(* PLC project CODESYS_HashTable_Struct_Example.project, CODESYS CODESYS V3.5 SP20 Patch 3 *)
(* stored: creationDateTime 2025-01-24T23:29:18.215425, modificationDateTime 2025-01-24T23:25:16.619379 *)

TYPE ST_Product : STRUCT
  id : STRING;  (* 製品ID *)
  name : STRING;  (* 製品名 *)
  width : UINT;  (* 幅 *)
  length : UINT;  (* 長さ *)
  height : UINT;  (* 高さ *)
END_STRUCT;
END_TYPE

(* values of E_ProductSettingState: Create: 新規作成; Edit: 編集 *)

{attribute 'qualified_only'}
{attribute 'strict'}
TYPE E_ProductSettingState : (Initial := 0, Create, Edit);
END_TYPE

INTERFACE IProductElement
PROPERTY ProductValue : ST_Product
END_PROPERTY
END_INTERFACE

PROGRAM PRG_ProductSetting
  VAR
    HashTableFactory : COL.HashTableFactory;  (* Factory to create a hash table on heap memory. *)
    productMap : COL.IMap3 := HashTableFactory.Create(udiMaxElements := 100);  (* Creates a hashtable on heap memory. NOTE: Collections that have been created with this Factory are not online change safe. *)
    productElementFactory : FB_ProductElementFactory;
    productNameArray : ARRAY[0..GVL.MAX_PRODUCT_NUM] OF STRING;  (* Visualizaton用 *)
    pnArrayLastIndex : UINT := 0;  (* 次に挿入する位置 *)
    state : E_ProductSettingState := E_ProductSettingState.Initial;
    selectedProductIndex : UINT;
    selectedProductId : STRING;
    visuProduct : ST_Product;
    msgBoxMessage : STRING;  (* メッセージBOX用 *)
    msgBoxEnabled : BOOL;
    msgBoxTap : BOOL;
    tmpValues : ARRAY[0..GVL.MAX_PRODUCT_NUM] OF ST_Product;  (* デバッグ用 *)
    iterator : COL.ListIterator;
    itfElement : COL.IElement;
    itfProductElement : IProductElement;
    xResult : BOOL;
    i : UINT;  (* 一時変数 *)
  END_VAR

                    //デバッグ用
i:=0;
productMap.Values(iterator);
WHILE iterator.HasNext() DO
	iterator.Next(itfElement=>itfElement);
	xResult := __QUERYINTERFACE(itfElement, itfProductElement);
	tmpValues[i] := itfProductElement.ProductValue;
	i:=i+1;
END_WHILE

//メッセージBOXを閉じる
IF msgBoxTap THEN
	msgBoxEnabled := FALSE;
	msgBoxTap := FALSE;
END_IF


//現在状態ごとの処理
IF state = E_ProductSettingState.Initial AND pnArrayLastIndex <> 0 THEN
	selectedProductIndex := 0;
	UpdateSelectedProduct();
	state := E_ProductSettingState.Edit;
END_IF
	

                  

METHOD DeleteProductFromNameArray
  VAR_INPUT
    info : ST_Product;
  END_VAR
  VAR
    i : UINT;
    deleteIndex : UINT;
    productId : STRING;
  END_VAR
                          IF pnArrayLastIndex > GVL.MAX_PRODUCT_NUM THEN
	RETURN;
END_IF


IF pnArrayLastIndex <> 0 THEN
	//昇順にソートされている前提で挿入個所を探索する
	FOR deleteIndex:=0 TO pnArrayLastIndex-1 DO
		productId := GetIdFromProductName(ADR(productNameArray[deleteIndex]));
		IF info.id = productId THEN
			productNameArray[deleteIndex] := '';
			EXIT;
		END_IF
	END_FOR
	
	//空いた箇所を詰める
	IF deleteIndex <> pnArrayLastIndex-1 THEN
		FOR i:=deleteIndex TO pnArrayLastIndex-1 DO
			productNameArray[i] := productNameArray[i+1];
		END_FOR
	END_IF
	
	productNameArray[pnArrayLastIndex-1] := '';
	pnArrayLastIndex := pnArrayLastIndex - 1;
	
END_IF

                        
END_METHOD

METHOD UpdateProductToNameArray
  VAR_INPUT
    info : ST_Product;
  END_VAR
  VAR
    concatStr : STRING;
    i : UINT;
    productId : STRING;
  END_VAR
                          IF pnArrayLastIndex > GVL.MAX_PRODUCT_NUM THEN
	RETURN;
END_IF

concatStr := CONCAT(info.id, '.');
concatStr := CONCAT(concatStr, info.name);

IF pnArrayLastIndex <> 0 THEN
	//昇順にソートされている前提で挿入個所を探索する
	FOR i:=0 TO pnArrayLastIndex-1 DO
		productId := GetIdFromProductName(ADR(productNameArray[i]));
		IF info.id = productId THEN
			productNameArray[i] := concatStr;
			EXIT;
		END_IF
	END_FOR
END_IF

                        
END_METHOD

METHOD DeleteProduct : BOOL
  VAR
    eError : COL.COLLECTION_ERROR;
    StringElementFactory : COL.StringElementFactory;  (* Factory to create StringElements on heap memory. *)
    concatStr : STRING;
  END_VAR
                          //表示中のデータを削除
eError := productMap.RemoveByKey(itfKey := StringElementFactory.Create(sValue := visuProduct.id));

//削除成功時
IF eError = COL.COLLECTION_ERROR.NO_ERROR THEN
	concatStr := CONCAT(visuProduct.id, '.');
	concatStr := CONCAT(concatStr, visuProduct.name);
	concatStr := CONCAT(concatStr, ' を削除しました');
	msgBoxMessage := concatStr;
	msgBoxEnabled := TRUE;
	//表示用Listの更新
	DeleteProductFromNameArray(visuProduct);
	ClearVisuProduct();
	state := E_ProductSettingState.Initial;
	
ELSE
	state := E_ProductSettingState.Initial;
END_IF;

                        
END_METHOD

METHOD Save : BOOL
  VAR
    eError : COL.COLLECTION_ERROR;
    contains : BOOL;
    StringElementFactory : COL.StringElementFactory;  (* Factory to create StringElements on heap memory. *)
    keyElement : COL.IStringElement;
    concatStr : STRING;
  END_VAR
                          keyElement := StringElementFactory.Create(sValue := visuProduct.id);
eError := productMap.ContainsKey(itfKey:=keyElement, xResult=>contains);

CASE state OF
	//更新時
	E_ProductSettingState.Edit:
		IF contains THEN
			
			eError := productMap.RemoveByKey(itfKey := keyElement);
			eError := productMap.AddKeyValuePair(itfKey := keyElement, itfValue := productElementFactory.Create(visuProduct));
			
			IF eError = COL.COLLECTION_ERROR.NO_ERROR THEN
				concatStr := CONCAT(visuProduct.id, '.');
				concatStr := CONCAT(concatStr, visuProduct.name);
				concatStr := CONCAT(concatStr, ' を更新しました');
				msgBoxMessage := concatStr;
				msgBoxEnabled := TRUE;
				UpdateProductToNameArray(visuProduct);
			ELSE
				msgBoxMessage := '更新に失敗しました。';
				msgBoxEnabled := TRUE;	
			END_IF
		END_IF
	
	//新規追加時
	E_ProductSettingState.Create:
		IF pnArrayLastIndex > GVL.MAX_PRODUCT_NUM-1 THEN
			msgBoxMessage := '登録可能な製品数の上限に達しています。';
			msgBoxEnabled := TRUE;
			RETURN;
		END_IF
		
		IF contains THEN
			msgBoxMessage := '既に同じIDが登録されています。別のIDをご使用ください。';
			msgBoxEnabled := TRUE;
			RETURN;
		END_IF
	
		eError := productMap.AddKeyValuePair(itfKey := keyElement, itfValue := productElementFactory.Create(visuProduct));
	
		IF eError = COL.COLLECTION_ERROR.NO_ERROR THEN
			concatStr := CONCAT(visuProduct.id, '.');
			concatStr := CONCAT(concatStr, visuProduct.name);
			concatStr := CONCAT(concatStr, ' を新規で追加しました');
			msgBoxMessage := concatStr;
			msgBoxEnabled := TRUE;
			//表示用Listの更新
			selectedProductIndex := InsertProductToNameArray(visuProduct);
			
			state := E_ProductSettingState.Edit;
			
		ELSE
			msgBoxMessage := '新規追加に失敗しました。';
			msgBoxEnabled := TRUE;
			state := E_ProductSettingState.Initial;
		END_IF
			
END_CASE


                        
END_METHOD

METHOD InsertProductToNameArray : UINT
  VAR_INPUT
    info : ST_Product;
  END_VAR
  VAR
    concatStr : STRING;
    insertIndex : UINT := 0;  (* 挿入個所のインデックス *)
    i : UINT;
  END_VAR
                          IF pnArrayLastIndex > GVL.MAX_PRODUCT_NUM-1 THEN
	RETURN;
END_IF

concatStr := CONCAT(info.id, '.');
concatStr := CONCAT(concatStr, info.name);


IF pnArrayLastIndex <> 0 THEN
	//昇順にソートされている前提で挿入個所を探索する
	FOR insertIndex:=0 TO pnArrayLastIndex-1 DO
		IF concatStr < productNameArray[insertIndex] THEN
			EXIT;
		END_IF
	END_FOR

	//挿入個所をあけるために1つずつずらす
	IF insertIndex <> pnArrayLastIndex THEN
		FOR i:=pnArrayLastIndex TO insertIndex+1 DO
			productNameArray[i] := productNameArray[i-1];
		END_FOR	
	END_IF
END_IF

productNameArray[insertIndex] := concatStr;
pnArrayLastIndex := pnArrayLastIndex + 1;

InsertProductToNameArray := insertIndex;
                        
END_METHOD

METHOD UpdateSelectedProduct
  VAR
    itfStringKey : COL.IStringElement;
    itfIInstance : FBF.IInstance;
    eError : COL.COLLECTION_ERROR;
    itfElement : COL.IElement;
    itfProductElement : IProductElement;
    selectedProductName : STRING;
    StringElementFactory : COL.StringElementFactory;  (* Factory to create StringElements on heap memory. *)
    xResult : BOOL;
  END_VAR
                          selectedProductName := productNameArray[selectedProductIndex];
selectedProductId := GetIdFromProductName(ADR(selectedProductName));
visuProduct := GetProductInfo(selectedProductId);
                        
END_METHOD

METHOD TransToCreateMode
                          state := E_ProductSettingState.Create;
selectedProductIndex := pnArrayLastIndex;

ClearVisuProduct();
                        
END_METHOD

METHOD CancelCreate
                          state := E_ProductSettingState.Initial;
selectedProductIndex := 0;
UpdateSelectedProduct();
                        
END_METHOD

METHOD SaveAs
                          state := E_ProductSettingState.Create;
selectedProductIndex := pnArrayLastIndex;
                        
END_METHOD

METHOD ClearVisuProduct
                          visuProduct.height := 0;
visuProduct.id := '';
visuProduct.length := 0;
visuProduct.name := '';
visuProduct.width := 0;
                        
END_METHOD

METHOD GetProductInfo : ST_Product
  VAR_INPUT
    id : STRING;
  END_VAR
  VAR
    itfStringKey : COL.IStringElement;
    itfIInstance : FBF.IInstance;
    eError : COL.COLLECTION_ERROR;
    itfElement : COL.IElement;
    itfProductElement : IProductElement;
    StringElementFactory : COL.StringElementFactory;  (* Factory to create StringElements on heap memory. *)
    xResult : BOOL;
  END_VAR
                          //MapからProductインスタンスを取得
itfStringKey := StringElementFactory.Create(sValue := id);
eError := productMap.GetElementByKey(itfKey := itfStringKey, itfValue => itfElement);
IF eError <> COL.COLLECTION_ERROR.NO_ERROR THEN
	RETURN;
END_IF

//キーの確認
xResult := __QUERYINTERFACE(itfStringKey, itfIInstance);
IF xResult THEN
	// Remove the temporary key
	itfIInstance.Dispose();
END_IF

//IElement形式からIProductElementに変換
xResult := __QUERYINTERFACE(itfElement, itfProductElement);
IF xResult THEN
	GetProductInfo := itfProductElement.ProductValue;
END_IF
                        
END_METHOD
END_PROGRAM

{attribute 'enable_dynamic_creation'}
{attribute 'hide'}
FUNCTION_BLOCK FB_Product EXTENDS FBF.InstanceData
  VAR_INPUT
    info : ST_PRODUCT;
  END_VAR

                    (* !! Do not add any executable code here !! *)
SUPER^();
                  
END_FUNCTION_BLOCK

(* Demo element with two integer values. An element must implement an interface which extends |COL.IElement|. This function block extends FBF.InstanceBase to enable dynamic creation via FBFactory. *)
{attribute 'no_explicit_call' := 'Explicit calls not allowed.'}
FUNCTION_BLOCK FB_ProductElement EXTENDS FBF.InstanceBase IMPLEMENTS IProductElement
  VAR_INPUT
    {attribute 'input_constant'}
    _product : ST_Product;
  END_VAR

                    
                  

(* Returns true of this element and itfElement are equal. This method will be called from the function block |COL.HashTable| to find an element by key if the hashcode of an element collides with an other element. IMPORTANT: The underlying value to be compared with MUST NOT be changed during the lifecycle of the object. *)
METHOD ElementEquals : BOOL
  VAR_INPUT
    itfElement : COL.IElement;  (* The element to compare *)
  END_VAR
  VAR
    element : IProductElement;
    xResult : BOOL;
    elementProduct : ST_Product;
    thisProduct : ST_Product;
  END_VAR
                          xResult := __QUERYINTERFACE(itfElement, element);
elementProduct := element.ProductValue;
thisProduct := ProductValue;
IF xResult THEN
	ElementEquals := thisProduct.id = elementProduct.id;	
ELSE
	ElementEquals := FALSE;
END_IF 
                        
END_METHOD

(* Returns the hashcode of this element. This method is used by hash based collections (e.g. |Hashtable|) to get the hashcode from a element. IMPORTANT: The value of the method MUST NOT be changed during the lifecycle of the object. *)
METHOD ElementHashCode : LINT
  VAR
    p : POINTER TO STRING;
  END_VAR
                          p := ADR(_product.id);
ElementHashCode := COL.HashCodeFromString(p);
                        
END_METHOD

(* Compares this element with itfElement. Returns 0 if the elements are equal, < 0 if the element is less than itfElement, > 0 if the element is greater than itfElement. This method will be called from sorted collections (e.g. |COL.SortedList|) to sort the elements. IMPORTANT: The underlying value to be compared with MUST NOT be changed during the lifecycle of the object. *)
METHOD ElementCompareTo : INT
  VAR_INPUT
    itfElement : COL.IElement;  (* The element to compare *)
  END_VAR
  VAR
    element : IProductElement;
    xResult : BOOL;
    elementProduct : ST_Product;
  END_VAR
                          // We use integer iInt1 for sorting.
xResult := __QUERYINTERFACE(itfElement, element);
IF xResult THEN
	elementProduct := element.ProductValue;
	IF _product.id < elementProduct.id THEN
		ElementCompareTo := -1;
	ELSIF _product.id > elementProduct.Id THEN
		ElementCompareTo := 1;
	ELSE
		ElementCompareTo := 0;
	END_IF
ELSE
	ElementCompareTo := -1;
END_IF 

                        
END_METHOD

(* This methode is called from the factory to give a chance to initialize the new fb instance with the content of itfData *)
METHOD prvInstInit : FBF.ERROR
  VAR_INPUT
    itfData : FBF.IData;
  END_VAR
  VAR
    pData : POINTER TO FB_Product;
    xOk : BOOL;
    thisProduct : ST_Product;
  END_VAR
                          SUPER^.prvInstInit(itfData);
xOk := __QUERYPOINTER(itfData, pData);
IF xOk THEN
	ProductValue := pData^.info;
END_IF

                        
END_METHOD

PROPERTY ProductValue : ST_Product
GET
                            ProductValue := _product;

                          
END_GET
SET
                            _product := ProductValue;

                          
END_SET
END_PROPERTY
END_FUNCTION_BLOCK

FUNCTION GetIdFromProductName : STRING
  VAR_INPUT
    productNamePtr : POINTER TO STRING;
  END_VAR

                    SplitString(productNamePtr, '.', sLeft=>GetIdFromProductName);
                  
END_FUNCTION

(* IElement factory for INT values *)
{attribute 'enable_dynamic_creation'}
FUNCTION_BLOCK FB_ProductElementFactory EXTENDS FBF.FactoryBase

                    SUPER^();

                  

(* Creates a IntElement *)
METHOD Create : IProductElement
  VAR_INPUT
    inputData : ST_Product;
  END_VAR
  VAR_OUTPUT
    eError : FBF.ERROR;
  END_VAR
  VAR
    hInst : CAA.HANDLE;
    itfInst : FBF.IInstance;
    xOk : BOOL;
    itfData : FB_Product;
    pInstance : POINTER TO FB_ProductElement;
  END_VAR
                          (* !!! This code must not be subject to change !!! *)
itfData(info:=inputData);
hInst := SUPER^.prvAllocInstMem(eError => eError);
pInstance := SUPER^.prvGetInstPointer(hInst);
IF pInstance <> 0 AND eError = FBF.ERROR.NO_ERROR THEN

	{implicit on}
	pInstance^.__vfInit();
	pInstance^.FB_Init(TRUE, FALSE);
	{implicit off}

	xOk := __QUERYINTERFACE(pInstance^, itfInst);
	IF xOk THEN
		xOk := SUPER^.prvInstInit(itfInst, hInst, itfData, eError=>eError);
	ELSE
		eError := FBF.ERROR.WRONG_INTERFACE;
	END_IF

	IF NOT xOk THEN
		SUPER^.prvFreeInstMem(hInst);
		Create := CAA.gc_pNULL;
    ELSE
        __QUERYINTERFACE(pInstance^, Create);
	END_IF
END_IF

                        
END_METHOD

(* {attribute 'conditionalshow' := 'SomeText'} {attribute 'conditionalshow'} {attribute 'hide'} *)
PROPERTY prvInstCount : CAA.COUNT
GET
                            (* Please choose a proper value for prvInstCount *)
prvInstCount := 10;
                          
END_GET
END_PROPERTY

(* {attribute 'conditionalshow' := 'SomeText'} {attribute 'conditionalshow'} {attribute 'hide'} *)
PROPERTY prvInstPoolExtendsFactor : USINT
GET
                            (* Please choose a proper value for prvInstPoolExtendsFactor *)
(* This value will be interpreted as a 0..x% size extendsion related to the original size of the pool *)
prvInstPoolExtendsFactor := 20;
                          
END_GET
END_PROPERTY

(* {attribute 'conditionalshow' := 'SomeText'} {attribute 'conditionalshow'} {attribute 'hide'} *)
PROPERTY prvInstSize : CAA.SIZE
GET
                            (* Please replace CustomFB with your specific function block type *)
prvInstSize := sizeof(FB_ProductElement);
                          
END_GET
END_PROPERTY
END_FUNCTION_BLOCK

CONFIGURATION Device
  RESOURCE Application ON PLC
    {attribute 'qualified_only'}
    VAR_GLOBAL CONSTANT  (* GVL *)
      MAX_PRODUCT_NUM : UINT := 100;
    END_VAR
    TASK MainTask(INTERVAL := T#20ms, PRIORITY := 1);
    TASK VISU_TASK(INTERVAL := T#100ms, PRIORITY := 31);
    PROGRAM PRG_ProductSetting WITH MainTask : PRG_ProductSetting;
    PROGRAM VisuElems.Visu_Prg WITH VISU_TASK : VisuElems.Visu_Prg;
  END_RESOURCE
END_CONFIGURATION
